(*
Nazwa:			P07_CapPusher
Opis:			Wvijak nasadek z sorteram wibracyjnym
Wersja:			v0.1
Data:			2025-11-03
Autor:			DP
Urzadzenia:		
Konfiguracja:	
Info:
- 
*)
PROGRAM P07_CapPusher
VAR_INPUT
	//Szlaban
	//...
	
	//Podajnik
	//...
	
	//Zakrecanie
	//..

END_VAR
VAR
	(*****************SZLABAN*******************)
	fbCapPusherGate										: FB_SpringGateV2;
	QbCapPusherGate										AT %Q*: BOOL; 			// Wyjście sterujące 

	(*******************PODAJNIK*********************)
	fbCapPusherFeeder									: FB_CapPusherFeeder;
	fbCapPusherFeederState								: FB_State;	
	eCapPusherFeederState								: E_Station;
	eCapPusherFeederRunningState						: E_CapFeederState; 	// Stan pracy 
	QbCapPusherFeederSorterVibrator 					AT %Q*: BOOL; 			// Wyjście sterujące 
	QbCapPusherFeederSorterVibrator2 					AT %Q*: BOOL; 			// Wyjście sterujące 	
	QbCapPusherFeederSorterAir 							AT %Q*: BOOL; 			// Wyjście sterujące 
	IbCapPusherFeederHopperSensor						: BOOL; 					
	IbCapPusherFeederWheelSensor						: BOOL; 			
	IbCapPusherFeederSleeveSensor					: BOOL; 
	QnCapPusherFeederVelocitySV 						AT %Q*: UDINT; 			// Nastawa prędkości
	InCapPusherFeederVelocityCV 						AT %I*: UDINT;		
	InCapPusherFeederSTW 								AT %I*: UINT; 			// Statusword transportera wejściowo wyjściowego
	QnCapPusherFeederCTW 								AT %Q*: UINT;  			// Controlword transportera we/wy
	IbCapPusherFeederWcState							AT %I*: BOOL; 			// Statusword transportera wejściowo wyjściowego
	TimerCapPusherFeederEnable							: TOF;
	rtCapPusherFeederEnable								: R_TRIG;
	tonCapPusherFeederEnable							: TON;
	
	(*******ZAKRECANIE**********)
	fbCapPusher											: FB_CapPusher;
	fbCapPusherState									: FB_State;	
	eCapPusherState										: E_Station;
	eCapPusherRunningState								: E_GripperScrewer; 	// Stan pracy 	

	QbCapPusher											AT %Q*: BOOL; 	
	QbCapPusherBlockActuator							AT %Q*: BOOL; 	
	QbCapPusherFormPositioning							AT %Q*: BOOL; 	
	
	IbCapPusherFormSensor								: BOOL; 
	IbCapPusherCapSensor								: BOOL; 
	IbCapPusherUpSensor									: BOOL; 
	IbCapPusherDownSensor								: BOOL; 
	IbCapPusherBlockActuatorOnSensor					: BOOL; 
	IbCapPusherBlockActuatorOffSensor					: BOOL; 
	IbCapPusherFormPositioningUpSensor					: BOOL; 
	IbCapPusherFormPositioningDownSensor				: BOOL; 
	TimerCapPusherEnable								: TOF;
	rtCapPusherEnable									: R_TRIG;
	tonCapPusherEnable									: TON;
	
	(*RFID*)
	//Przed
	bReadedCard 										: BOOL;				
	nReadedCard											: ULINT;	
	fbReader   											: FB_IfmIoLinkRfid;
	AusiReaderInputData  								AT %I* : ARRAY[0..27] OF USINT;
	IbReaderTagPresent									AT %I* : BOOL;
	IBReaderErrorValue									AT %I* : BYTE;
	IbReaderCmdEnd										AT %I* : BOOL;
	IBReaderDataCounterIn								AT %I* : BYTE;
	IbReaderCmdStartAck									AT %I* : BOOL;
	IbReaderCmdStart									AT %Q* : BOOL;
	IBReaderCmmandValue									AT %Q* : BYTE;
	IBReaderDataCounterOut								AT %Q* : BYTE;
	AusiReaderOutputData  								AT %Q* : ARRAY[0..27] OF USINT;	

	(*Lampy*)
	QbCapPusherRedSignalizationLamp 					AT %Q* : BOOL;				
	QbCapPusherGreenSignalizationLamp 					AT %Q* : BOOL;					
	QbCapPusherYellowSignalizationLamp 					AT %Q* : BOOL;							
	
	(*Przyciski*)

	(*Safety*)
		

	QbCapPusherDoors0Close								AT %Q* :BOOL;		// Rozkaz zamkniecia 
	
	(*Zawór główny*)
	QbCapPusherCompressedAir							AT %Q*		:BOOL;		
	IbCapPusherCompressedAirOK 							AT %I*		:BOOL;		//Zasilanie powietrzem sprężonym OK	
	
	(*Zasilanie*)
	IbCapPusherFuseFB1OK								AT %I* :BOOL;		//		
	IbCapPusherFuseFB2OK								AT %I* :BOOL;		//	
	IbCapPusherFuseFB3OK								AT %I* :BOOL;		//	
	
	(*DI wyspy pneumatycznej*)
	QABPneumaticCapPusherEB1ValveCoils 						AT %Q* 	: ARRAY[1..5] OF BYTE;	
	IABPneumaticCapPusherEB1DigitalInput 					AT %I* 	: ARRAY[1..4] OF BYTE;
	IuiPneumaticCapPusherEB1State							AT %I* 	: UINT;	

	(*Czujniki formatek*)
	IbCapPusherThirdFormSensor	 							: BOOL; 		// Czujnik dojazdu 3 formatki
	
	(*Manual*)
	
	(****Inne***)

	
END_VAR

aPowerSupply();
aButtons();
aPneumatics();
aRFID();
aRFID_FB();
aSafety();
aSignalization();
aLimits();
a1_Gate();
a1_GateTime();
a2_Feeder();
a3_Capping();
aWarnings();

(*BAZOWANIE - ZMIAN*)
//SSzlaban
//...
//Podajnik
tonCapPusherFeederEnable (IN:=bCapPusherEnable,PT:=T#5S); 
rtCapPusherFeederEnable(CLK:=tonCapPusherFeederEnable.Q,Q=>);
IF rtCapPusherFeederEnable.Q AND (P00_PackML.fbPMLAuto.ePMLState = E_PMLState.ePMLState_IDLE OR P00_PackML.fbPMLAuto.ePMLState = E_PMLState.ePMLState_EXECUTE)   THEN
	VIS_CP.bCapPusherFeederHeightSet:=TRUE;
ELSIF fbCapPusherFeeder.eState=E_Station.eHomingDone	OR	VIS.bErrorOccure THEN
 	VIS_CP.bCapPusherFeederHeightSet:=FALSE;
END_IF
//Zakrecanie
tonCapPusherEnable (IN:=bCapPusherEnable,PT:=T#5S); 
rtCapPusherEnable(CLK:=tonCapPusherEnable.Q,Q=>);
IF rtCapPusherEnable.Q AND (P00_PackML.fbPMLAuto.ePMLState = E_PMLState.ePMLState_IDLE OR P00_PackML.fbPMLAuto.ePMLState = E_PMLState.ePMLState_EXECUTE)   THEN
	VIS_CP.bCapPusherHeightSet:=TRUE;
ELSIF fbCapPusher.eState=E_Station.eHomingDone	OR	VIS.bErrorOccure THEN
 	VIS_CP.bCapPusherHeightSet:=FALSE;
END_IF
(*KONIEC BAZOWANIE - ZMIANA*)

(*Opoznienie wyłączanie enabla*)
//Szlaban
//..
//Podajnik
TimerCapPusherFeederEnable	(IN:=bCapPusherEnable,	PT:=T#2S);
//Zakrecanie
TimerCapPusherEnable		(IN:=bCapPusherEnable, PT:=T#2S);

(*Staty*)
//Szlaban
//...
//Podajnik
fbCapPusherFeederState(
	eState							:=	eCapPusherFeederState , 
	bRun							:=	VIS_CP.bCapPusherFeederRun,	
	eCapFeederRunningState			:=	eCapPusherFeederRunningState , 
	sStateDesc						=>	VIS_CP.sCapPusherFeederState,
	iState							=>	VIS_CP.iCapPusherFeederState);	

//Zakrecanie
fbCapPusherState(
	eState							:=	eCapPusherState , 
	bRun							:=	VIS_CP.bCapPusherRun,	
	eGripperScrewerRunningState		:=	eCapPusherRunningState , 
	sStateDesc						=>	VIS_CP.sCapPusherState,
	iState							=>	VIS_CP.iCapPusherState);	


(********KASOWANIE ROZKAZÓW CYKLI*********)
//Szlaban
//...
//Podajnik
//...
//Zakrecanie
IF fbCapPusher.bCycleDone1 AND bManualMode THEN
	VIS_CP.bCapPusherRun 		:= FALSE;
END_IF

ACTION a1_Gate:
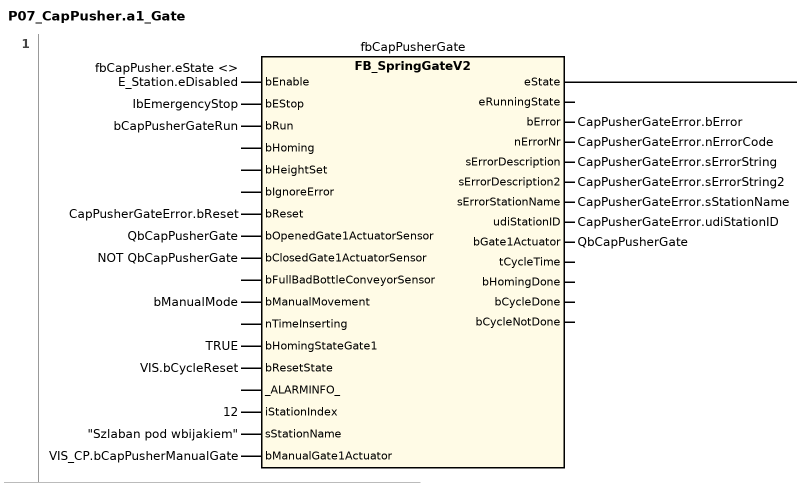
// NETWORK 1
fbCapPusherGate(
    bEnable := fbCapPusher.eState <> E_Station.eDisabled,
    bEStop := IbEmergencyStop,
    bRun := bCapPusherGateRun,
    bReset := CapPusherGateError.bReset,
    bOpenedGate1ActuatorSensor := QbCapPusherGate,
    bClosedGate1ActuatorSensor := NOT QbCapPusherGate,
    bManualMovement := bManualMode,
    bHomingStateGate1 := TRUE,
    bResetState := VIS.bCycleReset,
    iStationIndex := 12,
    sStationName := "Szlaban pod wbijakiem",
    bManualGate1Actuator := VIS_CP.bCapPusherManualGate,
    bError => CapPusherGateError.bError,
    nErrorNr => CapPusherGateError.nErrorCode,
    sErrorDescription => CapPusherGateError.sErrorString,
    sErrorDescription2 => CapPusherGateError.sErrorString2,
    sErrorStationName => CapPusherGateError.sStationName,
    udiStationID => CapPusherGateError.udiStationID,
    bGate1Actuator => QbCapPusherGate); // FB_SpringGateV2
END_ACTION

ACTION a1_GateTime:

fbCapPusherGate.nTimeInserting	:=	300;
END_ACTION

ACTION a2_Feeder:
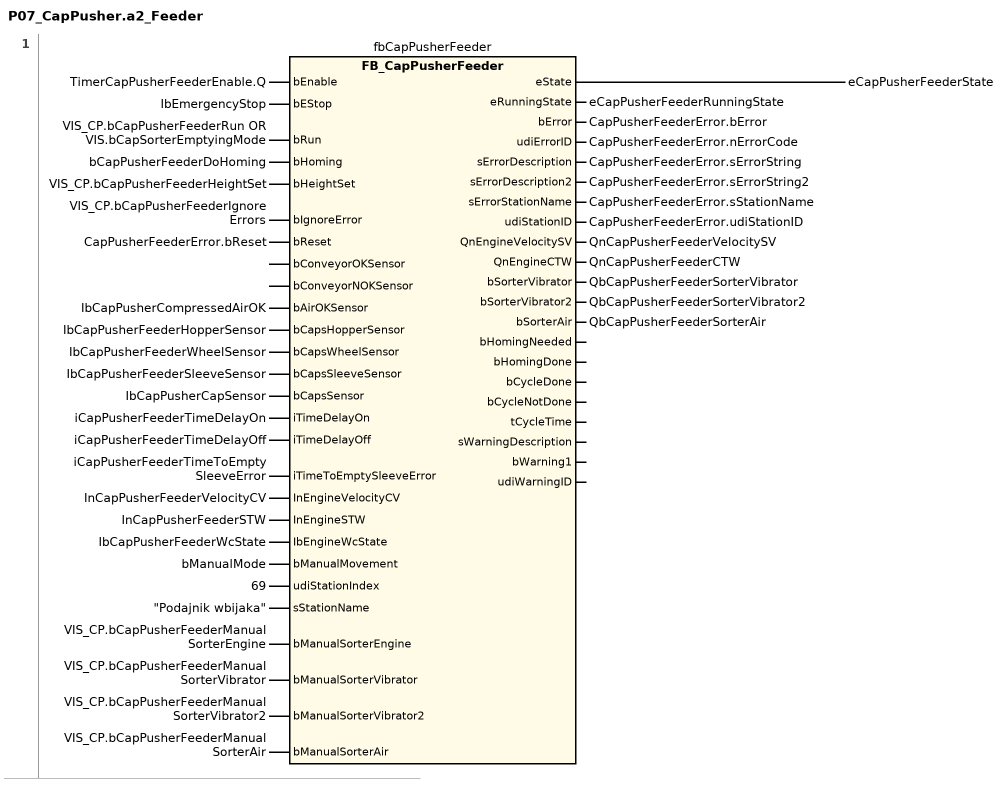
// NETWORK 1
fbCapPusherFeeder(
    bEnable := TimerCapPusherFeederEnable.Q,
    bEStop := IbEmergencyStop,
    bRun := VIS_CP.bCapPusherFeederRun OR VIS.bCapSorterEmptyingMode,
    bHoming := bCapPusherFeederDoHoming,
    bHeightSet := VIS_CP.bCapPusherFeederHeightSet,
    bIgnoreError := VIS_CP.bCapPusherFeederIgnoreErrors,
    bReset := CapPusherFeederError.bReset,
    bAirOKSensor := IbCapPusherCompressedAirOK,
    bCapsHopperSensor := IbCapPusherFeederHopperSensor,
    bCapsWheelSensor := IbCapPusherFeederWheelSensor,
    bCapsSleeveSensor := IbCapPusherFeederSleeveSensor,
    bCapsSensor := IbCapPusherCapSensor,
    iTimeDelayOn := iCapPusherFeederTimeDelayOn,
    iTimeDelayOff := iCapPusherFeederTimeDelayOff,
    iTimeToEmptySleeveError := iCapPusherFeederTimeToEmptySleeveError,
    InEngineVelocityCV := InCapPusherFeederVelocityCV,
    InEngineSTW := InCapPusherFeederSTW,
    IbEngineWcState := IbCapPusherFeederWcState,
    bManualMovement := bManualMode,
    udiStationIndex := 69,
    sStationName := "Podajnik wbijaka",
    bManualSorterEngine := VIS_CP.bCapPusherFeederManualSorterEngine,
    bManualSorterVibrator := VIS_CP.bCapPusherFeederManualSorterVibrator,
    bManualSorterVibrator2 := VIS_CP.bCapPusherFeederManualSorterVibrator2,
    bManualSorterAir := VIS_CP.bCapPusherFeederManualSorterAir,
    eRunningState => eCapPusherFeederRunningState,
    bError => CapPusherFeederError.bError,
    udiErrorID => CapPusherFeederError.nErrorCode,
    sErrorDescription => CapPusherFeederError.sErrorString,
    sErrorDescription2 => CapPusherFeederError.sErrorString2,
    sErrorStationName => CapPusherFeederError.sStationName,
    udiStationID => CapPusherFeederError.udiStationID,
    QnEngineVelocitySV => QnCapPusherFeederVelocitySV,
    QnEngineCTW => QnCapPusherFeederCTW,
    bSorterVibrator => QbCapPusherFeederSorterVibrator,
    bSorterVibrator2 => QbCapPusherFeederSorterVibrator2,
    bSorterAir => QbCapPusherFeederSorterAir); // FB_CapPusherFeeder
eCapPusherFeederState := fbCapPusherFeeder.eState;
END_ACTION

ACTION a3_Capping:
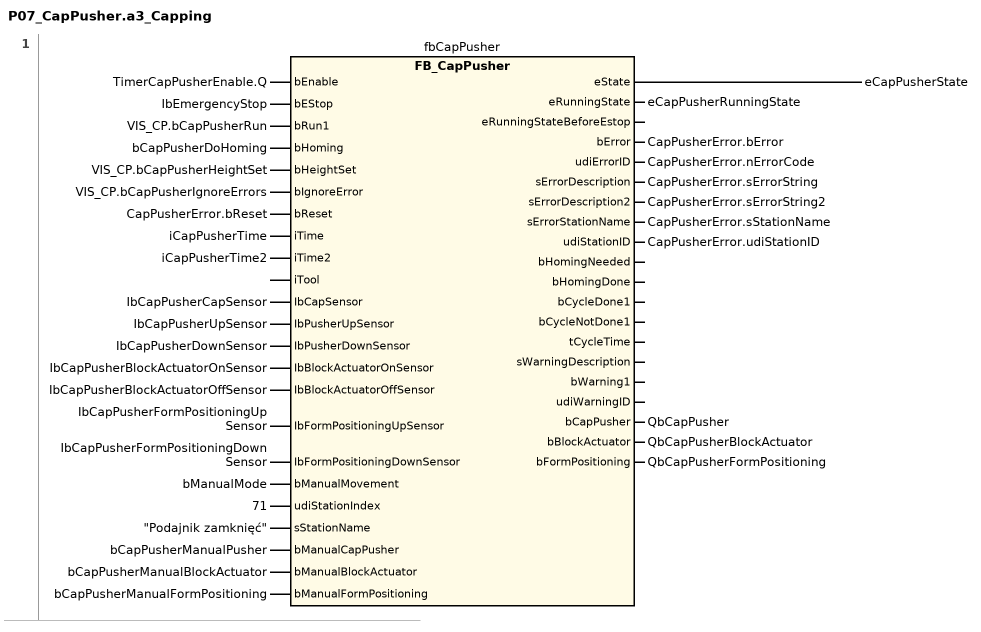
// NETWORK 1
fbCapPusher(
    bEnable := TimerCapPusherEnable.Q,
    bEStop := IbEmergencyStop,
    bRun1 := VIS_CP.bCapPusherRun,
    bHoming := bCapPusherDoHoming,
    bHeightSet := VIS_CP.bCapPusherHeightSet,
    bIgnoreError := VIS_CP.bCapPusherIgnoreErrors,
    bReset := CapPusherError.bReset,
    iTime := iCapPusherTime,
    iTime2 := iCapPusherTime2,
    IbCapSensor := IbCapPusherCapSensor,
    IbPusherUpSensor := IbCapPusherUpSensor,
    IbPusherDownSensor := IbCapPusherDownSensor,
    IbBlockActuatorOnSensor := IbCapPusherBlockActuatorOnSensor,
    IbBlockActuatorOffSensor := IbCapPusherBlockActuatorOffSensor,
    IbFormPositioningUpSensor := IbCapPusherFormPositioningUpSensor,
    IbFormPositioningDownSensor := IbCapPusherFormPositioningDownSensor,
    bManualMovement := bManualMode,
    udiStationIndex := 71,
    sStationName := "Podajnik zamknięć",
    bManualCapPusher := bCapPusherManualPusher,
    bManualBlockActuator := bCapPusherManualBlockActuator,
    bManualFormPositioning := bCapPusherManualFormPositioning,
    eRunningState => eCapPusherRunningState,
    bError => CapPusherError.bError,
    udiErrorID => CapPusherError.nErrorCode,
    sErrorDescription => CapPusherError.sErrorString,
    sErrorDescription2 => CapPusherError.sErrorString2,
    sErrorStationName => CapPusherError.sStationName,
    udiStationID => CapPusherError.udiStationID,
    bCapPusher => QbCapPusher,
    bBlockActuator => QbCapPusherBlockActuator,
    bFormPositioning => QbCapPusherFormPositioning); // FB_CapPusher
eCapPusherState := fbCapPusher.eState;
END_ACTION

ACTION aButtons:

END_ACTION

ACTION aLimits:
(*
Nazwa:			aLimits
Opis:			Zabezpieczenia
Wersja:			v1.0
Data:			2023-11-24
Autor:			DP
Urzadzenia:		
Zmiany:	

Info:
*)

(**** Limity i zabezpieczenia***)
END_ACTION

ACTION aPneumatics:
// Do podpięcia według kolejności
QbCapPusherGate;
QbCapPusherFeederSorterAir;
QbCapPusher;			
QbCapPusherBlockActuator;	
QbCapPusherFormPositioning;

(*************************** CapPusher EB1 **************************************)
// Wyspa 1 - dozowanie
IuiPneumaticCapPusherEB1State;
QABPneumaticCapPusherEB1ValveCoils[1].0	:= QbCapPusher;
QABPneumaticCapPusherEB1ValveCoils[1].1 := NOT QbCapPusher;
QABPneumaticCapPusherEB1ValveCoils[1].2 := QbCapPusherBlockActuator;
QABPneumaticCapPusherEB1ValveCoils[1].3 ;
QABPneumaticCapPusherEB1ValveCoils[1].4 := QbCapPusherFormPositioning;
QABPneumaticCapPusherEB1ValveCoils[1].5 ;
QABPneumaticCapPusherEB1ValveCoils[1].6 := NOT QbCapPusherGate;
QABPneumaticCapPusherEB1ValveCoils[1].7 := QbCapPusherGate; 
QABPneumaticCapPusherEB1ValveCoils[2].0 ;				
QABPneumaticCapPusherEB1ValveCoils[2].1 ;
QABPneumaticCapPusherEB1ValveCoils[2].2 ;
QABPneumaticCapPusherEB1ValveCoils[2].3 ;
QABPneumaticCapPusherEB1ValveCoils[2].4 ;											
QABPneumaticCapPusherEB1ValveCoils[2].5 ;
QABPneumaticCapPusherEB1ValveCoils[2].6 ;
QABPneumaticCapPusherEB1ValveCoils[2].7 ;
QABPneumaticCapPusherEB1ValveCoils[3].0 ;
QABPneumaticCapPusherEB1ValveCoils[3].1 ;
QABPneumaticCapPusherEB1ValveCoils[3].2 ;
QABPneumaticCapPusherEB1ValveCoils[3].3 ;
QABPneumaticCapPusherEB1ValveCoils[3].4 ; 
QABPneumaticCapPusherEB1ValveCoils[3].5 ;
QABPneumaticCapPusherEB1ValveCoils[3].6 ;
QABPneumaticCapPusherEB1ValveCoils[3].7 ;                                               
QABPneumaticCapPusherEB1ValveCoils[4].0	;		                                
QABPneumaticCapPusherEB1ValveCoils[4].1 ;                                       
QABPneumaticCapPusherEB1ValveCoils[4].2	;		                                
QABPneumaticCapPusherEB1ValveCoils[4].3 ;                                      
QABPneumaticCapPusherEB1ValveCoils[4].4 ;		                                
QABPneumaticCapPusherEB1ValveCoils[4].5 ;        
QABPneumaticCapPusherEB1ValveCoils[4].6 ;		
QABPneumaticCapPusherEB1ValveCoils[4].7 ; 
                                                              
(*********************Koniec CapPusher EB1 **************************************) 


//Zawór głównego powietrza
QbCapPusherCompressedAir	:=	IbEmergencyStop AND QbCapPusherFeederSorterAir;

(*************************** EB1 **************************************)
// Wyspa 1 - 52N8
IuiPneumaticCapPusherEB1State;
//DI1
IbCapPusherFeederHopperSensor		:=	IABPneumaticCapPusherEB1DigitalInput[1].0;	
IbCapPusherFeederWheelSensor		:=	NOT IABPneumaticCapPusherEB1DigitalInput[1].1;	
IbCapPusherFeederSleeveSensor		:=	IABPneumaticCapPusherEB1DigitalInput[1].2;	
										IABPneumaticCapPusherEB1DigitalInput[1].3;
IbCapPusherUpSensor					:=	IABPneumaticCapPusherEB1DigitalInput[1].4;	
IbCapPusherDownSensor				:=	IABPneumaticCapPusherEB1DigitalInput[1].5;	
IbCapPusherCapSensor				:=	IABPneumaticCapPusherEB1DigitalInput[1].6;	
										;IABPneumaticCapPusherEB1DigitalInput[1].7;	
//DI2                                           
IbCapPusherBlockActuatorOffSensor	:=	IABPneumaticCapPusherEB1DigitalInput[2].0;	
IbCapPusherBlockActuatorOnSensor	:=	IABPneumaticCapPusherEB1DigitalInput[2].1;	
IbCapPusherFormSensor				:=	IABPneumaticCapPusherEB1DigitalInput[2].2;	
IbCapPusherFormPositioningDownSensor:=	IABPneumaticCapPusherEB1DigitalInput[2].3;	
IbCapPusherFormPositioningUpSensor	:=	IABPneumaticCapPusherEB1DigitalInput[2].4;	
;	IABPneumaticCapPusherEB1DigitalInput[2].5;		
;	IABPneumaticCapPusherEB1DigitalInput[2].6;		
;	IABPneumaticCapPusherEB1DigitalInput[2].7;	

// Wyspa 1 - 52N8A
IuiPneumaticCapPusherEB1State;
//DI1
;	IABPneumaticCapPusherEB1DigitalInput[3].0;	
;	IABPneumaticCapPusherEB1DigitalInput[3].1;	
;	IABPneumaticCapPusherEB1DigitalInput[3].2;	
;	IABPneumaticCapPusherEB1DigitalInput[3].3;
;	IABPneumaticCapPusherEB1DigitalInput[3].4;	
;	IABPneumaticCapPusherEB1DigitalInput[3].5;		
;	IABPneumaticCapPusherEB1DigitalInput[3].6;		
;	IABPneumaticCapPusherEB1DigitalInput[3].7;
//DI2                                               		
;	IABPneumaticCapPusherEB1DigitalInput[4].0;
;	IABPneumaticCapPusherEB1DigitalInput[4].0;	
;	IABPneumaticCapPusherEB1DigitalInput[4].1;	
;	IABPneumaticCapPusherEB1DigitalInput[4].2;	
;	IABPneumaticCapPusherEB1DigitalInput[4].3;	
;	IABPneumaticCapPusherEB1DigitalInput[4].4;
;	IABPneumaticCapPusherEB1DigitalInput[4].5;		
;	IABPneumaticCapPusherEB1DigitalInput[4].6;		
	IABPneumaticCapPusherEB1DigitalInput[4].7;	
(*********************Koniec EB2 **************************************)
END_ACTION

ACTION aPowerSupply:


	//Dodane do głwnych
	IbCapPusherFuseFB1OK	; //Przekaznik kontroli faz
	IbCapPusherFuseFB2OK	; //Kontrola poprawności faz
	IbCapPusherFuseFB3OK	; //Blok bezpiecznikowy
END_ACTION

ACTION aRFID:
(*Przepisanie bity wykrycia karty*)
bReadedCard 		:= IbReaderTagPresent AND fbReader.bCodeReaded;
nReadedCard 		:= DINT_TO_ULINT(fbReader.diReadedCode);
END_ACTION

ACTION aRFID_FB:
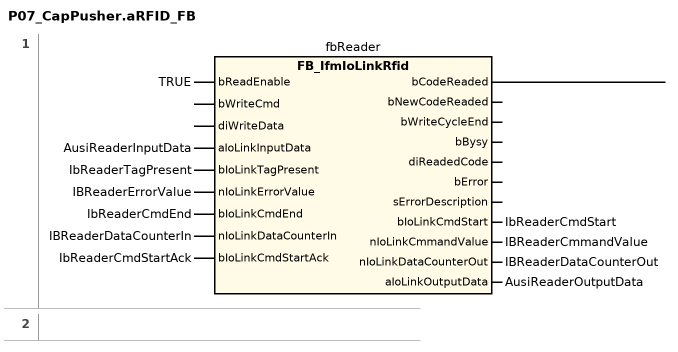
// NETWORK 1
fbReader(
    bReadEnable := TRUE,
    aIoLinkInputData := AusiReaderInputData,
    bIoLinkTagPresent := IbReaderTagPresent,
    nIoLinkErrorValue := IBReaderErrorValue,
    bIoLinkCmdEnd := IbReaderCmdEnd,
    nIoLinkDataCounterIn := IBReaderDataCounterIn,
    bIoLinkCmdStartAck := IbReaderCmdStartAck,
    bIoLinkCmdStart => IbReaderCmdStart,
    nIoLinkCmmandValue => IBReaderCmmandValue,
    nIoLinkDataCounterOut => IBReaderDataCounterOut,
    aIoLinkOutputData => AusiReaderOutputData); // FB_IfmIoLinkRfid

// NETWORK 2
END_ACTION

ACTION aSafety:

// Dodać do P00_Alarms.aGeneralAlarms
	//IbCapPusherEmergencyStopButton0Pressed;
	//IbCapPusherEmergencyStopButton1Pressed;
	
(*
	IF IbCapPusherEmergencyStopButton0Pressed THEN
		GeneralAlarms.nErrorCode:=1;			
		GeneralAlarms.sErrorString:='Stop Awaryjny, sprawdź bezpieczeństwo, zresetuj przyciskiem na panelu | Naciśnięty przycisk awaryjny 1 na CapPusher';	
	ELSIF  IbCapPusherEmergencyStopButton1Pressed THEN
		GeneralAlarms.nErrorCode:=2;
		GeneralAlarms.sErrorString:='Stop Awaryjny, sprawdź bezpieczeństwo, zresetuj przyciskiem na panelu | Naciśnięty przycisk awaryjny 2 na CapPusher';	
*)	
	

// Dodać do miejsca gdzie są zamykane drzwi	
// lub zostawić tak jak jest
	QbCapPusherDoors0Close := QbDispencersDoorsClose;
END_ACTION

ACTION aSignalization:
(*****Listwy LED*****)

QbCapPusherRedSignalizationLamp		:= INT_TO_BOOL(P00_Signalization.QiLineRedSignalizationLamp);
QbCapPusherGreenSignalizationLamp	:= INT_TO_BOOL(P00_Signalization.QiLineGreenSignalizationLamp);
QbCapPusherYellowSignalizationLamp	:= INT_TO_BOOL(P00_Signalization.QiLineBlueSignalizationLamp);


//QbCapPusherStartLamp	:= P00_Signalization.QbStartLamp;	   
//QbCapPusherResetLamp	:= P00_Signalization.QbResetLamp;
END_ACTION

ACTION aWarnings:
//Warning 0
IF fbCapPusherFeeder.bWarning1 AND NOT CapSorterWarning[0].bWarning THEN
	CapSorterWarning[0].bWarning										:=TRUE;
	CapSorterWarning[0].udiWarningCode									:=41;
	CapSorterWarning[0].sDescription									:='Sorter nasadek | Brak nasadek w zasobniku';
ELSIF NOT fbCapPusherFeeder.bWarning1 THEN 
	CapSorterWarning[0].bWarning										:=FALSE;
	CapSorterWarning[0].bAcknowledge									:=FALSE;
	VIS.uliWarningAcknowledge.27										:=FALSE;
ELSIF CapSorterWarning[0].bAcknowledge THEN                               
	CapSorterWarning[0].bAcknowledge									:=TRUE;
END_IF
END_ACTION

END_PROGRAM

(* stored: Version 1.2.0.0, ProductVersion 3.1.4026.13, FileIdentifier 760944b6afc0fe9f1aa37fa2ffa005e45768fbb4, FileSignature 2d974de3df2ed0b5da7c12242985b79e2e98a55a36e09ad7cd31172d16969fe111dd2d3ebfb596dc86678a9e6fec60cd58af327221aa18404a1027a66e4f06aede65e2a1f8fa81d33b76b702634c1cec46798a428749848ef2097787d9bdf0e431110f3add721a23e4e9c20dcc4e5029e7d8fdf7e03472bd8565e76e54a43ca9b7668875edfa584f45177288916062960526a68c59bea827ab2fcc4a9b538f7ecb302513086f47e10987b660688a102407fc2ba5e6e588d56ec978dfae640bad7b6515872a47c3d090af294725dc4de929e4af3f551c0185a3f4fa1b4eb3506da5399eb8a0ee343c127aca1a908d3505960685d4ac6284d66c7fb142184186ca
   POU P07_CapPusher: Id {59da9390-3c5c-41a2-9e70-94715a0417f7}, SpecialFunc None
   Action a1_Gate: Id {9fa45459-f65f-4e48-a5a6-92d585063e66}
   Action a1_GateTime: Id {4148e6b6-5e8a-4381-a447-b32cb6807cf6}
   Action a2_Feeder: Id {203a0d40-3f5d-4227-95f9-215e68247128}
   Action a3_Capping: Id {ee95d643-ea4a-44e0-a983-b16845eda513}
   Action aButtons: Id {9e7b798b-03bc-49ef-89d2-b46787872c1f}
   Action aLimits: Id {3e477bb6-5d98-406b-ad4b-5c266c8936ba}
   Action aPneumatics: Id {3111ec63-03ce-4941-a246-f79cc153bdd0}
   Action aPowerSupply: Id {6a0b1964-1a1e-4250-8079-9740f4f85bf4}
   Action aRFID: Id {0b036cf6-3249-4d3b-ac14-8793a84267c4}
   Action aRFID_FB: Id {14f04bca-40c8-4e3f-abbb-ddd206e2f41c}
   Action aSafety: Id {9509cb6f-459b-4197-8e9a-4442325a79f3}
   Action aSignalization: Id {deef0951-758a-4f74-a9da-5003eeb177c3}
   Action aWarnings: Id {72e43150-12e1-4533-bbf2-7607f8103608} *)
